// TIA Portal V16 export
// export: Created 2021-09-08T12:44:31.8339048Z, ExportSetting WithDefaults, DisplayName Totally Integrated Automation Portal, DisplayVersion V16 Update 3, DisplayName TIA Portal Version Control Interface, DisplayVersion V16 Update 2, DisplayName TIA Portal Openness, DisplayVersion V16 Update 3, DisplayName TIA Portal Teamcenter Gateway, DisplayVersion V16, DisplayName STEP 7 Professional, DisplayVersion V16 Update 3, DisplayName STEP 7 Safety, DisplayVersion V16, DisplayName WinCC Advanced, DisplayVersion V16 Update 3
VAR_GLOBAL   // PLC tag table "CONST"
END_VAR
VAR_GLOBAL CONSTANT   // user constants
   MAX_STEP_NUMB : Int := 50;
   MIN_STEP_NUMB : Int := 1;
   MAX_DEV_NUMB : Int := 16;
   MIN_DEV_NUMB : Int := 1;
   UF_CM_STANDBY : Int := 0;
   UF_CM_FILTRATION : Int := 2;
   UF_CM_START : Int := 1;
   UF_CM_HW : Int := 4;
   UF_CM_HW_A : Int := 5;
   UF_CM_CEB1 : Int := 6;
   UF_CM_CEB1_A : Int := 7;
   UF_CM_CEB2 : Int := 8;
   UF_CM_CEB2_A : Int := 9;
   UF_CM_STOP : Int := 3;
END_VAR
